{attribute 'pack_mode' := '1'}
TYPE TMachineSafety :
STRUCT
	bCanLockDoor		: BOOL;
	bLockDoor			: BOOL;
	bCanUnlockDoor		: BOOL;
	bUnlockDoor			: BOOL;
END_STRUCT
END_TYPE

(* stored: Version 1.1.0.1, ProductVersion 3.1.4022.12
   DUT TMachineSafety: Id {72a88380-f502-4055-af23-b748fdc75ad5} *)
